Fanuc KAREL source: NC0049.KL

-- PROVISIONAL review KL for V1013-1; original PC SHA256 74bb6dba7c1f627ece6415bd3ec17ee7156fd7697714a5fdebf2179396e1148a
-- Incomplete behavior may be omitted. Consult companion uncertainty JSON. Do not deploy.
PROGRAM NC0049
%NOLOCKGROUP
-- UNRESOLVED_LOCAL_POOL 1 cells at code offset 3; source declarations unknown
-- DIRECT_LOCAL_WORD_ACCESS alone does not prove INTEGER, REAL, or BOOLEAN
BEGIN
  -- UNRESOLVED_PC offsets 0-8; opcodes 2B,2C,7B
  -- UNRESOLVED_PC offsets 13-20; opcodes 9D,23
  -- UNRESOLVED_PC offsets 25-38; opcodes 21,9D,57,79
  -- UNRESOLVED_PC offsets 43-60; opcodes 21,40,41,42
  -- UNRESOLVED_PC offsets 65-78; opcodes 21,9D,57,79
  -- UNRESOLVED_PC offsets 83-100; opcodes 21,40,41,42
  -- UNRESOLVED_PC offsets 105-118; opcodes 21,9D,57,79
  -- UNRESOLVED_PC offsets 123-140; opcodes 21,40,41,42
  -- UNRESOLVED_PC offsets 145-158; opcodes 21,9D,57,79
  -- UNRESOLVED_PC offsets 163-180; opcodes 21,40,41,42
  -- UNRESOLVED_PC offsets 185-198; opcodes 21,9D,57,79
  -- UNRESOLVED_PC offsets 203-220; opcodes 21,40,41,42
  -- UNRESOLVED_PC offsets 225-238; opcodes 21,9D,57,79
  -- UNRESOLVED_PC offsets 243-260; opcodes 21,40,41,42
  -- UNRESOLVED_PC offsets 265-278; opcodes 21,9D,57,79
  -- UNRESOLVED_PC offsets 283-300; opcodes 21,40,41,42
  -- UNRESOLVED_PC offsets 305-318; opcodes 21,9D,57,79
  -- UNRESOLVED_PC offsets 323-337; opcodes 21,9D,52,23
  -- UNRESOLVED_PC offsets 342-347; opcodes 7A
  -- UNRESOLVED_PC offsets 352-370; opcodes 21,2E,52,23
  -- UNRESOLVED_PC offsets 375-391; opcodes 7A,40,41,42
  -- UNRESOLVED_PC offsets 396-420; opcodes 21,2E,52,23,7A,43
  -- UNRESOLVED_PC offsets 425-443; opcodes 21,2E,52,23
  -- UNRESOLVED_PC offsets 453-458; opcodes 7A
  -- UNRESOLVED_PC offsets 463-481; opcodes 21,2E,52,23
  -- UNRESOLVED_PC offsets 486-502; opcodes 7A,40,41,42
  -- UNRESOLVED_PC offsets 507-531; opcodes 21,2E,52,23,7A,43
  -- UNRESOLVED_PC offsets 536-554; opcodes 21,2E,52,23
  -- UNRESOLVED_PC offsets 564-569; opcodes 7A
  -- UNRESOLVED_PC offsets 574-592; opcodes 21,2E,52,23
  -- UNRESOLVED_PC offsets 597-613; opcodes 7A,40,41,42
  -- UNRESOLVED_PC offsets 618-642; opcodes 21,2E,52,23,7A,43
  -- UNRESOLVED_PC offsets 647-665; opcodes 21,2E,52,23
  -- UNRESOLVED_PC offsets 675-680; opcodes 7A
  -- UNRESOLVED_PC offsets 685-703; opcodes 21,2E,52,23
  -- UNRESOLVED_PC offsets 708-724; opcodes 7A,40,41,42
  -- UNRESOLVED_PC offsets 729-753; opcodes 21,2E,52,23,7A,43
  -- UNRESOLVED_PC offsets 758-776; opcodes 21,2E,52,23
  -- UNRESOLVED_PC offsets 786-791; opcodes 7A
  -- UNRESOLVED_PC offsets 796-814; opcodes 21,2E,52,23
  -- UNRESOLVED_PC offsets 819-835; opcodes 7A,40,41,42
  -- UNRESOLVED_PC offsets 840-864; opcodes 21,2E,52,23,7A,43
  -- UNRESOLVED_PC offsets 869-887; opcodes 21,2E,52,23
  -- UNRESOLVED_PC offsets 897-902; opcodes 7A
  -- UNRESOLVED_PC offsets 907-925; opcodes 21,2E,52,23
  -- UNRESOLVED_PC offsets 930-946; opcodes 7A,40,41,42
  -- UNRESOLVED_PC offsets 951-975; opcodes 21,2E,52,23,7A,43
  -- UNRESOLVED_PC offsets 980-998; opcodes 21,2E,52,23
  -- UNRESOLVED_PC offsets 1008-1013; opcodes 7A
  -- UNRESOLVED_PC offsets 1018-1036; opcodes 21,2E,52,23
  -- UNRESOLVED_PC offsets 1041-1057; opcodes 7A,40,41,42
  -- UNRESOLVED_PC offsets 1062-1086; opcodes 21,2E,52,23,7A,43
  -- UNRESOLVED_PC offsets 1091-1109; opcodes 21,2E,52,23
  -- UNRESOLVED_PC offsets 1119-1124; opcodes 7A
  -- UNRESOLVED_PC offsets 1129-1147; opcodes 21,2E,52,23
  -- UNRESOLVED_PC offsets 1157-1161; opcodes 7F
  -- UNRESOLVED_PC offsets 1166-1170; opcodes 27,AA
  -- UNRESOLVED_PC offsets 1175-1179; opcodes 7F
END NC0049
